FUNCTION_BLOCK mainGUIFB (* JADE WORKER *)
  (* Standard: 61499-1 *)
  (* Version 1.0, 2014-04-22, Ahmed, Fraunhofer IGD *)
  (* Compiler header: package fb.rt; *)
  (* Compiler Java Sun JDK 1.5.0 *)
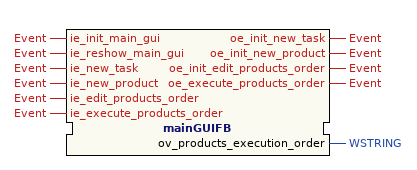
  EVENT_INPUT
    ie_init_main_gui;
    ie_reshow_main_gui;
    ie_new_task;
    ie_new_product;
    ie_edit_products_order;
    ie_execute_products_order;
  END_EVENT
  EVENT_OUTPUT
    oe_init_new_task;
    oe_init_new_product;
    oe_init_edit_products_order;
    oe_execute_products_order;
  END_EVENT
  VAR_OUTPUT
    ov_products_execution_order : WSTRING;
  END_VAR
END_FUNCTION_BLOCK
